Omron CX-Programmer project NewProject (CX-Programmer 9.75)

# PLC Yess1: CP1L M

## Global symbols (name address type ; comment)
0.00 BOOL  ; PB1
100.00 BOOL  ; Lamp
200.00 BOOL  ; M0
200.01 BOOL  ; M1
200.02 BOOL  ; M2
200.03 BOOL  ; M3
200.04 BOOL  ; M4

## Program NewProgram1 (cyclic task 0)
; Ahyar Mustafa Sangat Ganteng

### Section Section1

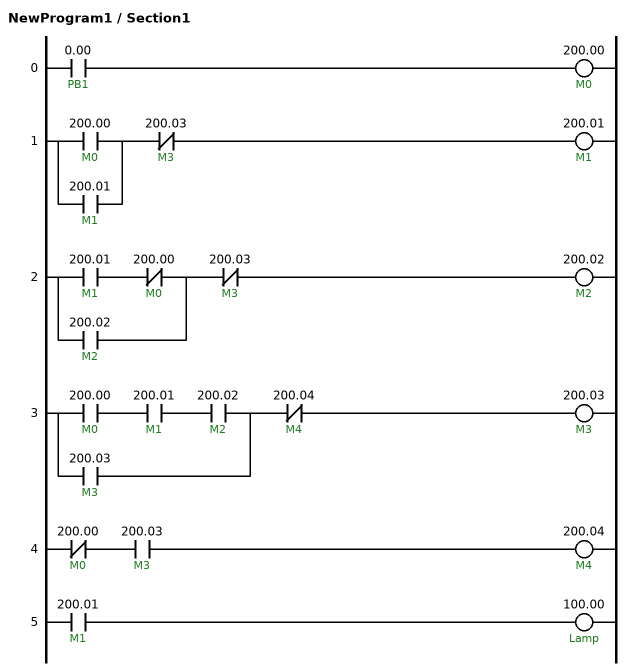
; rung 0
LD 0.00  ; PB1
OUT 200.00  ; M0
; rung 1
LD 200.00  ; M0
OR 200.01  ; M1
ANDNOT 200.03  ; M3
OUT 200.01  ; M1
; rung 2
LD 200.01  ; M1
ANDNOT 200.00  ; M0
OR 200.02  ; M2
ANDNOT 200.03  ; M3
OUT 200.02  ; M2
; rung 3
LD 200.00  ; M0
AND 200.01  ; M1
AND 200.02  ; M2
OR 200.03  ; M3
ANDNOT 200.04  ; M4
OUT 200.03  ; M3
; rung 4
LDNOT 200.00  ; M0
AND 200.03  ; M3
OUT 200.04  ; M4
; rung 5
LD 200.01  ; M1
OUT 100.00  ; Lamp

### Section END
; rung 0
END(001)